INTERFACE InterfaceObservableBase

END_INTERFACE

(* stored: Version 1.1.0.1, ProductVersion 3.1.4024.15
   Itf InterfaceObservableBase: Id {75016919-f109-4b6f-881f-ff3b2fc201c4} *)
